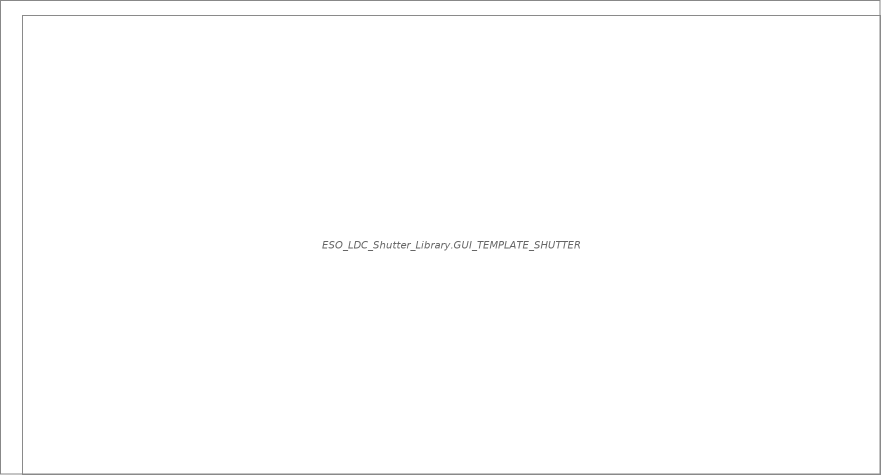
VISUALIZATION shutter1  // 881x475
    Frame (22,15 859x460)
        shows ESO_LDC_Shutter_Library.GUI_TEMPLATE_SHUTTER(m_Instance := MAIN.Shutter1)
END_VISUALIZATION

(* stored: Version 1.1.0.1, ProductVersion 3.1.4024.3
   Visu shutter1: Id {e4dbc4ef-2185-4208-a6f9-4aa55eade7e8} *)
